// TIA Portal V20 export
DATA_BLOCK "HMI_AlarmData"   // DB20220
{ S7_Optimized_Access := 'TRUE' }
// stored: AutoNumber false, MemoryReserve 100
   VAR
      "Word" : Array[0..7] of Word;
   END_VAR
BEGIN
   // "Word"[0] : MES
END_DATA_BLOCK
